FUNCTION_BLOCK FB_LamparaTemporizada_LD
VAR_INPUT
    TiempoEncendido: REAL := 2.0;
END_VAR
VAR_OUTPUT
    TiempoPendiente: REAL;
END_VAR
VAR
    Lampara AT %Q*: BOOL;
    Pulsador AT %I*: BOOL;
    
    Temporizador: TON;
    Memoria: RS;
    
    Resultado: REAL;
    Tiempo: TIME;
END_VAR

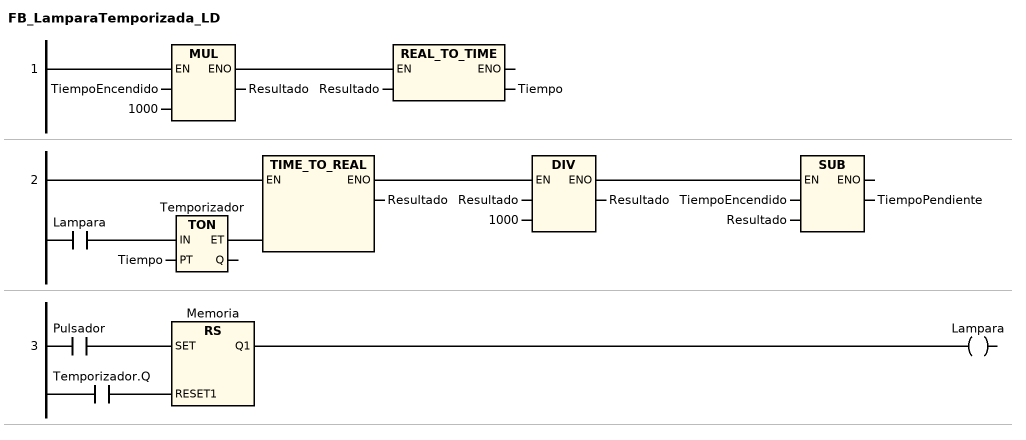
// NETWORK 1
Resultado := TiempoEncendido * 1000;
Tiempo := REAL_TO_TIME(Resultado);

// NETWORK 2
Temporizador(IN := Lampara, PT := Tiempo); // TON
Resultado := TIME_TO_REAL(Temporizador.ET);
Resultado := Resultado / 1000;
TiempoPendiente := TiempoEncendido - Resultado;

// NETWORK 3
Memoria(SET := Pulsador, RESET1 := Temporizador.Q); // RS
Lampara := Memoria.Q1;

END_FUNCTION_BLOCK

(* stored: Version 1.1.0.1, ProductVersion 3.1.4024.12
   POU FB_LamparaTemporizada_LD: Id {424061ba-8d78-48c7-b4ae-26f15978acd8}, SpecialFunc None *)
